(*
SPDX-FileCopyrightText: © 2026 Oleksandr Tiutyk <trofimich@gmail.com>
SPDX-License-Identifier: MIT
License: https://opensource.org/license/mit
*)

{attribute 'no_explicit_call' := 'do not call this function block directly'} 
{attribute 'enable_dynamic_creation'}
FUNCTION_BLOCK WhileActivity EXTENDS SequenceActivity IMPLEMENTS IWhileActivity
VAR
	{attribute 'OPC.UA.DA' := '0'}
	_ClassName_ : STRING := __POUNAME();

	{attribute 'OPC.UA.DA' := '0'}
	_Condition : ICondition;	
END_VAR

{attribute 'monitoring' := 'call'}
PROPERTY ClassName : REFERENCE TO STRING
GET
ClassName REF= _ClassName_;
END_GET
END_PROPERTY

{attribute 'monitoring' := 'call'}
PROPERTY FINAL Condition : ICondition
GET
Condition := _Condition;
END_GET
SET
_Condition := Condition;
END_SET
END_PROPERTY

METHOD Configure
VAR_INPUT
	condition : ICondition; 
END_VAR
VAR
	argumentNullException : TOF_Core.ArgumentNotSpecifiedException;
END_VAR
IF condition = 0 THEN
	argumentNullException.Throw(NamespaceName, ClassName, __POUNAME(), __POSITION(), 'condition');
END_IF

condition.ParentActivity := THIS^;

_Condition := condition;
END_METHOD

{attribute 'monitoring' := 'call'}
PROPERTY NamespaceName : REFERENCE TO STRING
GET
NamespaceName REF= CurrentNamespace.Name;
END_GET
END_PROPERTY

METHOD PROTECTED OnRunning : ACTIVITY_RUNNING_STATE
VAR_INPUT
	startRunning : BOOL;
	startResuming : BOOL;
END_VAR
VAR_OUTPUT
	haltReason : WSTRING(255);
END_VAR
VAR
	activity : IActivity;
	
	currentActivityIsNullException : TOF_Core.NullReferenceException;
END_VAR
VAR
	workflowVariable : TOF_Core.GENERIC_VALUE;
	
	argumentNullException : TOF_Core.NullReferenceException;
END_VAR
IF _Condition = 0 THEN
	argumentNullException.Throw(NamespaceName, ClassName, __POUNAME(), __POSITION(), 'Condition');
END_IF

activity := CurrentActivity;

IF startRunning OR_ELSE (startResuming AND_THEN activity = 0) THEN
	IF NOT _Condition.Evaluate(THIS^) THEN
		OnRunning := ACTIVITY_RUNNING_STATE.WORK_COMPLETED;
		RETURN;
	END_IF
END_IF

OnRunning := SUPER^.OnRunning(startRunning, startResuming, haltReason => haltReason);

IF OnRunning = ACTIVITY_RUNNING_STATE.WORK_COMPLETED AND_THEN _Condition.Evaluate(THIS^) THEN
	OnRunning := SUPER^.OnRunning(TRUE, FALSE, haltReason => haltReason);
END_IF
END_METHOD

{attribute 'monitoring' := 'call'}
PROPERTY SelfSize : ULINT
GET
SelfSize := XSIZEOF(THIS^);
END_GET
END_PROPERTY

END_FUNCTION_BLOCK

(* stored: Version 1.1.0.1
   POU WhileActivity: Id {a1dc987f-676e-48f4-8437-6b262709e26c}, SpecialFunc None
   Property ClassName: Id {e8c310a9-25a5-40fb-af06-20c97f669e26}
   Get Get: Id {9c476135-c2c6-4e6b-963b-cf0d4c8a0c66}
   Property Condition: Id {1569931e-587f-4563-a5bc-90730247f2a7}
   Get Get: Id {99562b20-36d6-457b-8c31-a7b8437d4df1}
   Set Set: Id {1ff2bd01-f001-40dc-ba83-6a4797b5f804}
   Method Configure: Id {977f0425-c37b-4e6b-8b39-b78bbd4d800a}
   Property NamespaceName: Id {86bb5599-d10e-42fb-95c9-1264df59ae02}
   Get Get: Id {8a7a6027-3e8c-4f60-888c-7717a6b92a11}
   Method OnRunning: Id {f271eeb4-f3d7-4733-877e-04b96312cb2b}
   Property SelfSize: Id {2c9eb82d-325f-4688-b541-736efe376418}
   Get Get: Id {9f76a8d8-910f-4548-8eb4-705d5ff59a56} *)
